// Mitsubishi GX Works2 project: 서보 모터 연습   PLC: Q03UDV

PROGRAM MAIN
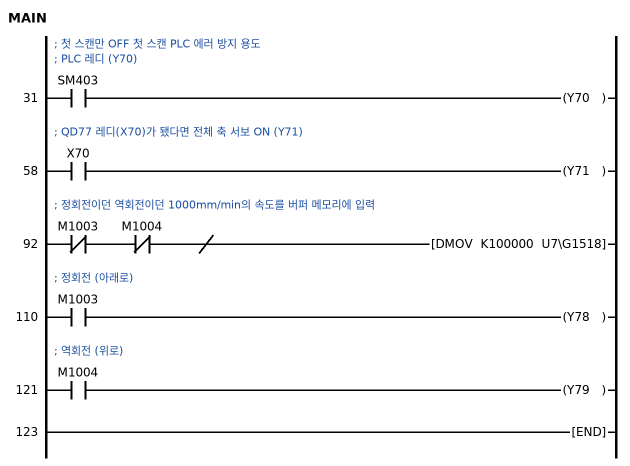
; 첫 스캔만 OFF 첫 스캔 PLC 에러 방지 용도
; PLC 레디 (Y70)
31    LD      SM403
      OUT     Y70
; QD77 레디(X70)가 됐다면 전체 축 서보 ON (Y71)
58    LD      X70
      OUT     Y71
; 정회전이던 역회전이던 1000mm/min의 속도를 버퍼 메모리에 입력
92    LDI     M1003
      ANI     M1004
      INV
      DMOV    K100000 U7\G1518
; 정회전 (아래로)
110   LD      M1003
      OUT     Y78
; 역회전 (위로)
121   LD      M1004
      OUT     Y79
123   END
END_PROGRAM
